TEXTLIST tlDetectionTunel
  0 = 'Initialization'
  3 = 'First Taring'
  5 = 'Checking '
  10 = 'Waiting for next step'
  15 = 'Going back with actuator'
  20 = 'Checking bottle weight'
  25 = 'Turning on conveyor and pushing out bottle'
  30 = 'Bottle was push'
  35 = 'Pushing actuator went back'
  70 = 'Botle pushout'
  75 = 'Bottle pushed out'
  80 = 'Actuator went back'
  90 = 'Error steps'
  91 = 'Waiting for reset'
  95 = 'Performing reset'
  17 = 'Vision sensor detection'
  18 = 'Vision sensor wait for end of work'
   = ''
END_TEXTLIST

(* stored: Version 1.1.0.1, ProductVersion 3.1.4024.13
   TextList tlDetectionTunel: Id {15d20005-2972-4a5a-a8b9-b43a2ed18f32} *)
